FUNCTION_BLOCK StopTask EXTENDS TcoCore.TcoTask IMPLEMENTS ITcoDriveSimple
VAR
    {attribute addProperty Name "<#Deceleration#>"}
    _deceleration : LREAL;
    {attribute addProperty Name "<#Jerk#>"}
    _jerk : LREAL;
END_VAR
VAR
    {attribute 'hide'}
    _axisRef : REFERENCE TO TcoAxisRef;
    {attribute 'hide'}
    _mcStop : Tc2_MC2.MC_Stop;
END_VAR

IF NOT __ISVALIDREF(_axisRef) THEN
    IF __ISVALIDREF(DriveRef) THEN
        _axisRef REF= DriveRef.AxisRef;
    ELSE
        RETURN;
    END_IF
END_IF

IF THIS^.Ready OR THIS^.Done THEN
    _mcStop(Axis := _axisRef, Execute := FALSE);
END_IF

IF THIS^.State = TcoCore.eTaskState.Requested THEN
    //In case of error, drive  is reseted first.
    IF THIS^.DriveRef._axisRef.Status.Error THEN
        THIS^.DriveRef.Reset();
        RETURN;
        // When drive input is enabled, but MC_Power.Status has not yet reached value true, this condition postpone execution 
        //to ensure that movement is not triggered before drive is powered up. 
    ELSIF THIS^.DriveRef.inEnable AND NOT THIS^.DriveRef._axisStatus.Operational THEN
        RETURN;
    END_IF
END_IF

IF Execute() THEN
    _mcStop(Axis := _axisRef,
        Execute := NOT _mcStop.Busy,
        Deceleration := _deceleration,
        Jerk := _jerk,
        Done =>,
        Busy =>,
        Active =>,
        CommandAborted =>,
        Error =>,
        ErrorID =>);

    IF _mcStop.CommandAborted THEN
        THIS^.Abort();
    END_IF

    DoneWhen(_mcStop.Done);
    ThrowWhen(_mcStop.Error);
END_IF

PROPERTY DriveRef : REFERENCE TO TcoDriveSimple
GET
VAR
    _drive : ITcoDriveSimple := 0;
END_VAR
IF __QUERYINTERFACE(THIS^._Parent, _drive) THEN
    DriveRef REF= _drive.DriveRef;
END_IF
END_GET
END_PROPERTY

METHOD PUBLIC FB_init : BOOL
VAR_INPUT
    bInitRetains : BOOL; // if TRUE, the retain variables are initialized (warm start / cold start)
    bInCopyCode : BOOL; // if TRUE, the instance afterwards gets moved into the copy code (online change)
    Parent : ITcoObject;
END_VAR
SUPER^.FB_init(	bInitRetains	:=	bInitRetains,
				bInCopyCode		:=	bInCopyCode,	
				Parent			:=	Parent);
END_METHOD

METHOD INTERNAL InvokeWithParams : ITcoTaskStatus
VAR_INPUT
    inDeceleration : LREAL;
    inJerk : LREAL;
END_VAR
_deceleration := inDeceleration;
_jerk := inJerk;
InvokeWithParams := THIS^.Invoke();
END_METHOD

(*~
	<docu>
		<summary>
			Restores this instance to the Ready state. Can be called explicitly or from within one of the restore mechanisms.
			<para>
				See also <see cref="TcoTask.PlcTcoTask.AutoRestorable()"/>
			</para>
		</summary>			
	</docu>	
~*)
METHOD Restore : ITcoRestorable
SUPER^.Restore();
END_METHOD

END_FUNCTION_BLOCK

(* stored: Version 1.1.0.1, ProductVersion 3.1.4024.6
   POU StopTask: Id {74d9043e-4117-01d9-3a62-1eb57ed666eb}, SpecialFunc None
   Property DriveRef: Id {9b09ccb4-872f-0610-145e-0f12d134830d}
   Get Get: Id {7837dcdc-9ef2-02df-3ea8-2c4ce8461cd5}
   Method FB_init: Id {602d6098-db54-0ea0-0640-8cf967f0aeae}
   Method InvokeWithParams: Id {c0055189-f8d8-0731-3212-5e2c8124424f}
   Method Restore: Id {60f9bd15-fddc-0be4-0113-68a2b17125e1} *)
